// TwinCAT 3 PLC project MainPLCProject
// ProgramVersion: 3.1.4024.0
// libraries:
//   Tc2_Standard, * (Beckhoff Automation GmbH)
//   Tc2_System, * (Beckhoff Automation GmbH)
//   Tc2_TcpIp, * (Beckhoff Automation GmbH)
//   Tc2_Utilities, * (Beckhoff Automation GmbH)
//   Tc3_Module, * (Beckhoff Automation GmbH)
//   VisuDialogs, * (System)
//   VisuSymbols,3.5.10.0,System
// project tree:
//   DUTs/ ClientState.TcDUT, COM_MODE.TcDUT, DataExchangeState.TcDUT, Command.TcDUT, Message.TcDUT, MessageLogData.TcDUT, ReceiveStatus.TcDUT, SendStatus.TcDUT
//   / GlobalTextList.TcGTLO, PlcTask.TcTTO, Visualization Manager.TcVMO (not stored)
//   GVLs/ GVL.TcGVL, GVL_Constants.TcGVL
//   POUs/Classes/ ClientDataExchanger.TcPOU, COMMUNICATION.TcPOU, MESSAGE_CREATOR.TcPOU, MESSAGE_HANDLER.TcPOU, TCPClient.TcPOU
//   POUs/Helpers/ AddCounterToMessage.TcPOU, LogToWarning.TcPOU, ShiftHistoryLeft.TcPOU
//   POUs/ MAIN.TcPOU
//   VISUs/ VisualizationControlPanel.TcVIS
// real-time tasks:
//   TASK PlcTask: cycle T#10ms, priority 20, ADS port 350
//   TASK HeartbeatTask: cycle T#50000us, priority 1, ADS port 351

CONFIGURATION MainPLCProject
    RESOURCE PLC ON TwinCAT3
        TASK PlcTask(INTERVAL := T#10ms, PRIORITY := 20);
        PROGRAM MAIN WITH PlcTask : MAIN;
    END_RESOURCE
END_CONFIGURATION

// ---- DUTs/ClientState.TcDUT
{attribute 'qualified_only'}
{attribute 'strict'}
TYPE ClientState :
(
	IDLE,
	SENDING,
	RECEIVING
) := IDLE;
END_TYPE

// ---- DUTs/COM_MODE.TcDUT
{attribute 'qualified_only'}
{attribute 'strict'}
TYPE COM_MODE :
(
	Robot,
	Monarco
);
END_TYPE

// ---- DUTs/DataExchangeState.TcDUT
{attribute 'qualified_only'}
{attribute 'strict'}
TYPE DataExchangeState :
(
	IDLE,
	START,
	WORKING,
	ERROR
) := START;
END_TYPE

// ---- DUTs/Command.TcDUT
TYPE Command :
STRUCT CONSTANT
	Start : STRING(9) := 'CRISTART';
	End : STRING(7) := 'CRIEND';
	MovementVar : STRING(4) := 'VAR';
	Heartbeat : STRING(9) := 'ALIVEJOG';
	
END_STRUCT
END_TYPE

// ---- DUTs/Message.TcDUT
// Pre-made robot messages
TYPE Message :
STRUCT CONSTANT
	Connect : STRING(30) := 'CMD Connect';
	AliveDemo : STRING(63) := 'ALIVEJOG 40.0 50.0 40.0 30.0 30.0 0.0 0.0 0.0 0.0';	//Do not use, only for testing!
	EnableMessage : STRING(80) := 'CMD Enable';
END_STRUCT
END_TYPE

// ---- DUTs/MessageLogData.TcDUT
TYPE MessageLogData :
STRUCT
	systemTimeString : T_MaxString := '';
	message : STRING(GVL_Constants.MAX_RECEIVE_MESSAGE_LENGTH) := '';
END_STRUCT
END_TYPE

// ---- DUTs/ReceiveStatus.TcDUT
{attribute 'qualified_only'}
{attribute 'strict'}
TYPE ReceiveStatus :
(
	WAITING,
	RECEIVING,
	DONE,
	FAIL,
	TIMEOUT
) := RECEIVING;
END_TYPE

// ---- DUTs/SendStatus.TcDUT
{attribute 'qualified_only'}
{attribute 'strict'}
TYPE SendStatus :
(
	SENDING,
	FAIL,
	SUCCESS
) := SENDING;
END_TYPE

// ---- GVLs/GVL.TcGVL
{attribute 'qualified_only'}
VAR_GLOBAL
	// COMMUNICATION variables
	ReceivedStringArray : ARRAY[0..200] OF STRING;
	ReceivedStringWordCounter : INT := 0;

	ReceivedCMD : STRING := '';
	VarValue : STRING := '';
	VarType : STRING := '';
	VarName : STRING := '';
	//
END_VAR

// ---- GVLs/GVL_Constants.TcGVL
{attribute 'qualified_only'}
VAR_GLOBAL CONSTANT
	MAX_RECEIVE_MESSAGE_LENGTH : UDINT := 1024;
	MAX_HISTORY_SIZE : BYTE := 10;
END_VAR

// ---- POUs/MAIN.TcPOU
PROGRAM MAIN
VAR CONSTANT
	LOCAL_IP : T_IPv4Addr := '127.0.0.1';
	LOCAL_PORT : UDINT := 8080;

	REMOTE_IP : T_IPv4Addr := '192.168.3.1';
	REMOTE_PORT : UDINT := 8080;
	
	ROBOT_IP : T_IPv4Addr := '192.168.3.11';
	ROBOT_PORT : UDINT := 3920;
	
	command : Command := ();
	message : Message := ();
	//endHistoryIndex : BYTE := 9;

END_VAR
VAR
	buttonConnectPressed : BOOL;
	buttonDisconnectPressed : BOOL;	
	buttonSendPressed : BOOL;
	buttonConnectToRobotPressed : BOOL;
	buttonDebugSendPressed : BOOL;
	buttonEnableMotorsPressed : BOOL;
	
	connectTrigger : R_TRIG;
	disconnectTrigger : R_TRIG;
	sendTrigger : R_TRIG;
	connectToRobotTrigger : R_TRIG;
	debugSendTrigger : R_TRIG;
	enableMotorsTrigger : R_TRIG;
	
	client : TCPClient(LOCAL_IP, LOCAL_PORT, isEnabled := FALSE);
	LocalSystemTime : FB_LocalSystemTime;
	
	// COMMUNICATION message handling
	MessageBase : COMMUNICATION(CommunicationMODE := COM_MODE.Monarco);
	messageHandler : MESSAGE_HANDLER();
	MessageERROR : int := 0;
	//
	
	connectionMessage : STRING(20) := 'Disconnected';
	isHeartbeatEnabled : BOOL := FALSE;
	
	closeAllConnections : FB_SocketCloseALL();
	closeAll : BOOL := TRUE;	//Close all on initial startup
	
	//messageToServer : T_MaxString := 'CRISTART 1 CMD Connect CRIEND';
	messageToServer : T_MaxString := 'Hello world 2.0 CRIEND';
	debugMessageToServer : T_MaxString := 'VAR Joint 0.0 0.0 0.0 0.0 0.0 0.0 0.0 0.0 0.0';
	messageFromServer : STRING(GVL_Constants.MAX_RECEIVE_MESSAGE_LENGTH) := '';
	//finalSendMsg : STRING(100);
	
	heartbeatTimer : TON;
	heartbeatInterval : TIME := T#1S;
	
	sendCounter : INT := 1;
	finalAliveMessage : STRING(100) := '';
	totalMessagesFromServerCount : UDINT := 0;
	
	//TODO: Extract into fb? Separate task?
	currentTime : TIMESTRUCT;
	messageHistoryArray : ARRAY [0.. GVL_Constants.MAX_HISTORY_SIZE - 1] OF MessageLogData;
	currentHistoryIndex : BYTE := 0;
	currentMessageLogData : MessageLogData;
	
	//Testing
	
	executed : BOOL := FALSE;
	test : UDINT;
	test2 : UDINT;
	test3 : UDINT;

END_VAR

//On PLC reset/program download, close all connections
IF (closeAll) THEN	
	closeAll := FALSE;
	closeAllConnections(sSrvNetId := '', bExecute := TRUE, tTimeout := T#10S);
ELSE
	closeAllConnections(bExecute := FALSE);
END_IF

IF (closeAllConnections.bBusy) THEN
	RETURN;	//Do not continue the program until all connections are closed
END_IF

// === ===

// === UI Handling ===
LocalSystemTime(bEnable := TRUE, tTimeout := T#1S, systemTime => currentTime);

connectTrigger(CLK := buttonConnectPressed);
disconnectTrigger(CLK := buttonDisconnectPressed);
sendTrigger(CLK := buttonSendPressed);
connectToRobotTrigger(CLK := buttonConnectToRobotPressed);
debugSendTrigger(CLK := buttonDebugSendPressed);
enableMotorsTrigger(CLK := buttonEnableMotorsPressed);

IF (client.IsConnected) THEN
	connectionMessage := 'Connected';
ELSE
	connectionMessage := 'Disconnected';
END_IF

IF (connectTrigger.Q) THEN
	CASE MessageBase.COMMUNICATION_MODE OF
	// check for communication mode and set IP for this mode.
		COM_MODE.Robot:
			client.RemoteServerAddress := LOCAL_IP;
			client.RemoteServerPort := LOCAL_PORT;
		
		COM_MODE.Monarco:
			client.RemoteServerAddress := ROBOT_IP;
			client.RemoteServerPort := ROBOT_PORT;
	END_CASE
	client.BindReceiveMessage(variableToBind := messageFromServer);
	client.Enable();
END_IF

IF (disconnectTrigger.Q) THEN
	client.Disable();
END_IF

// === Message Sending ===
CASE MessageBase.COMMUNICATION_MODE OF
	COM_MODE.Robot:
// ROBOT COM
		IF (sendTrigger.Q) THEN  // debug: send move command to robot.
			client.Send(messageToSend := MessageBase.CREATE(COMMAND := 'VAR', COMMAND_DETAILS := 'Joint 0.0 0.0 0.0 0.0 0.0 0.0 0.0 0.0 0.0', ERROR => MessageERROR));
		END_IF

		IF (debugSendTrigger.Q) THEN // debug: not in use jet.
			client.Send(messageToSend := MessageBase.CREATE(COMMAND := '', COMMAND_DETAILS := '', ERROR => MessageERROR));
		END_IF

		IF (connectToRobotTrigger.Q) THEN
			client.Send(messageToSend := MessageBase.CREATE(COMMAND := 'CMD', COMMAND_DETAILS := 'Connect', ERROR => MessageERROR));
			isHeartbeatEnabled := TRUE;
		END_IF

		IF (enableMotorsTrigger.Q) THEN
			client.Send(messageToSend := MessageBase.CREATE(COMMAND := 'CMD', COMMAND_DETAILS := 'Enable', ERROR => MessageERROR));
		END_IF
//		
	COM_MODE.Monarco:
// MONARCO COM
		IF (sendTrigger.Q) THEN 
			client.Send(messageToSend := MessageBase.CREATE(COMMAND := 'CMD', COMMAND_DETAILS := 'LED_ON', ERROR => MessageERROR));
		END_IF

		IF (debugSendTrigger.Q) THEN
			client.Send(messageToSend := MessageBase.CREATE(COMMAND := 'CMD', COMMAND_DETAILS := 'LED_OFF', ERROR => MessageERROR));
		END_IF
//
END_CASE

// === Message Receiving ===
IF (client.NewMessageAvailable(clearFlag := TRUE)) THEN
	//Update history
	IF (currentHistoryIndex >= GVL_Constants.MAX_HISTORY_SIZE) THEN
		//Ran out of history space, discard youngest member
		currentHistoryIndex := GVL_Constants.MAX_HISTORY_SIZE;
		ShiftHistoryLeft(arr := messageHistoryArray);
	ELSE
		//Can still append
		currentHistoryIndex := currentHistoryIndex + 1;
	END_IF
	
	//Handle message
	MessageBase.HANDLE(messageFromServer);
	
	//Add new entry
	currentMessageLogData.message := messageFromServer;	
	currentMessageLogData.systemTimeString := SYSTEMTIME_TO_STRING(in := currentTime);
	messageHistoryArray[currentHistoryIndex - 1] := currentMessageLogData;
END_IF
// === ===

// === Heartbeat ===
heartbeatTimer(IN := isHeartbeatEnabled, PT := heartbeatInterval);

IF (heartbeatTimer.Q AND client.IsClientEnabled) THEN
	heartbeatTimer(IN := FALSE);
	client.Send(messageToSend := MessageBase.CREATE('ALIVEJOG', '40.0 50.0 40.0 30.0 30.0 0.0 0.0 0.0 0.0', ERROR => MessageERROR));
END_IF
// === ===

client(totalMessagesReceived => totalMessagesFromServerCount);

END_PROGRAM

// ---- POUs/Classes/TCPClient.TcPOU
FUNCTION_BLOCK TCPClient
VAR CONSTANT
	CLIENT_RECONNECT_TIME : TIME := T#31S;
	MAX_MESSAGE_LENGTH : INT := 255;
	MAX_RECEIVE_MESSAGE_LENGTH : UDINT := GVL_Constants.MAX_RECEIVE_MESSAGE_LENGTH;
END_VAR
VAR_OUTPUT
	totalMessagesReceived : UDINT := 0;
END_VAR
VAR
	m_isClientEnabled : BOOL := TRUE;	
	m_serverNetID : STRING(80) := '';
	
	ClientServerConnection : FB_ClientServerConnection;
	SocketSend : FB_SocketSend;
	SocketReceive : FB_SocketReceive;
	m_clientDataExchanger : ClientDataExchanger;	//Note implemented yet: leave for later, use as
	m_socketHandle : T_HSOCKET;
	
	
	m_remoteServerAddress : T_IPv4Addr;	
	m_remoteServerPort : UDINT := 0;
	
	//Note: make it an input and send only when the class is called?
	m_messageToSend : T_MaxString := 'Hello world!';
	//m_messageReceived : T_MaxString;	// The latest message received from the server //TODO: REMOVE, Depricated
	m_messageReceivedRef : REFERENCE TO STRING(MAX_RECEIVE_MESSAGE_LENGTH);
	
	m_isConnected : BOOL := FALSE;
	m_isBusy : BOOL;
	m_errorOccured : BOOL;
	m_lastErrorId : UDINT;
	
	
	m_currentSocketState : Tc2_TcpIp.E_SocketConnectionState;
	m_currentState : ClientState := ClientState.RECEIVING;	

	m_sendDataExchangeState : DataExchangeState := DataExchangeState.START;	
	m_sendRequested: BOOL;
	m_sendStatus : SendStatus;
	m_sendErrorId : UDINT;
	m_sendTimeout : TIME := T#15S;	//Note: Lower?
	
	//Receiving
	m_receiveDataExchangeState : DataExchangeState := DataExchangeState.IDLE;	
	m_isReceiveTimerEnabled : BOOL := TRUE;
	m_receiveTimer : TON();
	m_isReceiveTimeoutEnabled : BOOL := FALSE;	
	m_receiveTimeoutTimer : TON();
	m_receiveBuffer : STRING(MAX_RECEIVE_MESSAGE_LENGTH) := '';
	m_totalBytesReceived : UDINT := 0;
	m_receiveTimeout : TIME := T#1M;
	m_readInterval : TIME := T#10MS;
//	m_receiveMessageDelimiter : BYTE := F_ToASC(';');	//Note: Use plain 0 (without F_ToASC()) for \0
	m_receiveMessageDelimiter : BYTE := 0;	//'\0'	//Not used currently
	m_delimiterString : STRING(80) := 'CRIEND';	//TODO: Make settable via property
	m_receivedMessage : T_MaxString := '';
	m_receiveStatus : ReceiveStatus;
	m_newDataAvailable : BOOL := FALSE;	//Reset to false when it is read
	m_receiveErrorId : UDINT := 0;
	m_totalMessagesReceived : UDINT := 0;
END_VAR

//Handler code
//Does that need to be executed every cycle or can I put it in eSOCKET_DISCONNECTED state?
ClientServerConnection(sSrvNetID := m_serverNetID,
						 nMode := 0,
						 sRemoteHost := RemoteServerAddress,
						 nRemotePort := m_remoteServerPort,
						 tReconnect := CLIENT_RECONNECT_TIME,
						 bEnable := IsClientEnabled,
						 bBusy => m_isBusy,
						 bError => m_errorOccured,
						 nErrId => m_lastErrorId,
						 hSocket => m_socketHandle,
						 eState => m_currentSocketState);

CASE m_currentSocketState OF
	E_SocketConnectionState.eSOCKET_DISCONNECTED:
		m_isConnected := FALSE;
	//
	E_SocketConnectionState.eSOCKET_SUSPENDED:
	//Change from disconnected to connected or vise versa
		m_isConnected := FALSE;
	//
	E_SocketConnectionState.eSOCKET_CONNECTED:
		m_isConnected := TRUE;
END_CASE

IF (NOT m_isConnected) THEN
	RETURN;
END_IF

// Executed only if a connection is established

CASE m_currentState OF
	//
	ClientState.SENDING:
		m_sendStatus := SendMessage(messageToSend := m_messageToSend, timeout := m_sendTimeout, errorId => m_sendErrorId);
		IF (m_sendStatus = SendStatus.SUCCESS) THEN
			m_currentState := ClientState.RECEIVING;
		ELSIF (m_sendStatus = SendStatus.FAIL) THEN
			//Sending failed
			ADSLOGDINT(msgCtrlMask := ADSLOG_MSGTYPE_WARN, msgFmtStr := 'Send fail error: %d', dintArg := UDINT_TO_DINT(m_sendErrorId));
			m_currentState := ClientState.RECEIVING;
		END_IF
		
	//
	ClientState.RECEIVING:
		m_receiveStatus := Receive(timeout := m_receiveTimeout, 
									readInterval := m_readInterval, 
									messageDelimiter := m_receiveMessageDelimiter,	//Currently not used
									errorId => m_receiveErrorId);
		
		IF (m_receiveStatus <> ReceiveStatus.RECEIVING) THEN
			IF (m_receiveStatus = ReceiveStatus.DONE) THEN
				//
				totalMessagesReceived := totalMessagesReceived + 1;
				m_newDataAvailable := TRUE;
			END_IF
			
			IF (m_receiveStatus = ReceiveStatus.FAIL) THEN
				//Fail Handling
				LogToWarning(msgFmtStr := 'Receive fail error: %s', messageArg := UDINT_TO_STRING(m_receiveErrorId));
			END_IF
			
			IF (m_receiveStatus = ReceiveStatus.TIMEOUT) THEN
				//Timeout handling
				LogToWarning(msgFmtStr := 'Receive timed out', messageArg := '');
				//Disable();	//Disable on timeout
			END_IF
	
			IF (m_sendRequested) THEN
				m_sendRequested := FALSE;
				m_sendErrorId := 0;
				m_currentState := ClientState.SENDING;
			END_IF
		END_IF						
	
	// After done receiving, go to idle?
	//
END_CASE

METHOD PUBLIC BindReceiveMessage : BOOL
VAR_INPUT
	variableToBind : REFERENCE TO STRING(MAX_RECEIVE_MESSAGE_LENGTH);
END_VAR
m_messageReceivedRef REF= variableToBind;
END_METHOD

METHOD PUBLIC Disable : BOOL
m_isClientEnabled := False;
END_METHOD

METHOD PUBLIC Enable : BOOL
VAR_INPUT
END_VAR
m_isClientEnabled := TRUE;
END_METHOD

METHOD FB_init : BOOL
VAR_INPUT
	bInitRetains : BOOL; // if TRUE, the retain variables are initialized (warm start / cold start)
	bInCopyCode : BOOL;  // if TRUE, the instance afterwards gets moved into the copy code (online change)
	
	remoteServerAddress : T_IPv4Addr := '127.0.0.1';
	remoteServerPort : UDINT := 8080;
	isEnabled : BOOL := FALSE;
END_VAR
m_remoteServerAddress := remoteServerAddress;
m_remoteServerPort := remoteServerPort;
m_isClientEnabled := isEnabled;
END_METHOD

PROPERTY IsClientEnabled : BOOL
GET
IsClientEnabled := m_isClientEnabled;
END_GET
END_PROPERTY

PROPERTY IsConnected : BOOL
GET
IsConnected := m_isConnected;
END_GET
END_PROPERTY

PROPERTY LastSendStatus : SendStatus
GET
LastSendStatus := m_sendStatus;
END_GET
END_PROPERTY

METHOD PUBLIC NewMessageAvailable : BOOL
VAR_INPUT
	clearFlag : BOOL := FALSE;	//Clears the new message flag if set to true, does not otherwise
END_VAR
NewMessageAvailable := m_newDataAvailable;

IF (clearFLag) THEN
	m_newDataAvailable := FALSE;
END_IF
END_METHOD

METHOD PRIVATE Receive : ReceiveStatus
VAR_INPUT
	timeout : TIME := T#10S;
	readInterval : TIME := T#10MS;
	messageDelimiter : BYTE := 0;
END_VAR

VAR_OUTPUT
	errorId : UDINT;
END_VAR

VAR
	errorOccurred : BOOL;	//can sty
	isBusy : BOOL;	//can stay																
	
	timedout : BOOL := FALSE;	//Output of TON
	receivedBytes : UDINT := 0;	//Output, should be fine to be here
	
	startPosition : UDINT := 0;	//Can stay, assigned before used
	endPosition : UDINT := 0;	//Can stay, assigned before used
	currentFrameLength : UDINT := 0; // Length of string received this cycle	//Should be fine
	posOfDelimiter : UDINT := 0;
	
	
	index : UDINT := 0;	//For-loop index
	
END_VAR
m_receiveTimer(IN := m_isReceiveTimerEnabled);
m_receiveTimeoutTimer(IN := m_isReceiveTimeoutEnabled, PT := timeout, Q => timedout);

CASE m_receiveDataExchangeState OF
	DataExchangeState.IDLE:
		//Reset variables
		m_isReceiveTimerEnabled := FALSE;
		m_receiveTimer(IN := m_isReceiveTimerEnabled, PT := T#0MS); 	//Do not wait for the first read
		m_isReceiveTimeoutEnabled := FALSE;
		Receive := ReceiveStatus.WAITING;
		m_receiveDataExchangeState := DataExchangeState.START;
	//
	DataExchangeState.START:
		Receive := ReceiveStatus.WAITING;
		m_isReceiveTimerEnabled := TRUE;
		IF (m_receiveTimer.Q) THEN
			SocketReceive(bExecute := FALSE);
			SocketReceive(sSrvNetId := m_serverNetID,
						  hSocket := m_socketHandle,
						  pDest := ADR(m_receiveBuffer) + m_totalBytesReceived,
						  cbLen := SIZEOF(m_receiveBuffer) - m_totalBytesReceived,
						  tTimeout := timeout,
						  bExecute := TRUE);	
			
			m_receiveDataExchangeState := DataExchangeState.WORKING;
		END_IF
	//
	DataExchangeState.WORKING:
		Receive := ReceiveStatus.RECEIVING;
		SocketReceive(bExecute := FALSE,
				tTimeout := timeout,
				bBusy => isBusy,
				bError => errorOccurred,
				nErrId => errorId,
				nRecBytes => receivedBytes);
		//Enable timeout
		IF (NOT isBusy AND NOT errorOccurred) THEN
			IF (receivedBytes > 0) THEN
				startPosition := m_totalBytesReceived;
				//Calculate new total
				m_totalBytesReceived := m_totalBytesReceived + receivedBytes;
				endPosition := m_totalBytesReceived - 1;
				currentFrameLength := 0;
				//Only proceed if we have enough space
				IF (m_totalBytesReceived < SIZEOF(m_messageReceivedRef)) THEN
					m_receiveTimer (PT := T#0MS); //Read asap
					//Bytes received, disable timeout check
					m_isReceiveTimeoutEnabled := FALSE;
					//Search for end of message delimiter
					posOfDelimiter := INT_TO_UDINT(FIND(STR1 := m_receiveBuffer, STR2 := m_delimiterString));
					
					IF (posOfDelimiter = 0) THEN
						//Delimiter not found
						LogToWarning('Delim not found', '');
						RETURN;
					END_IF
					
					currentFrameLength := posOfDelimiter + 6{delimiter size} - 1;
					MEMCPY(destAddr := ADR(m_messageReceivedRef), srcAddr := ADR(m_receiveBuffer), n := currentFrameLength);
					MEMSET(destAddr := ADR(m_receiveBuffer), fillByte := 0, n := SIZEOF(m_receiveBuffer));	//Clear buffer
					m_totalBytesReceived := 0;
					
					//All received
					Receive := ReceiveStatus.DONE;
					m_receiveDataExchangeState := DataExchangeState.IDLE;
					//OLD Find TODO: Find a way to implement via a function? So that you can use both
//					FOR index := startPosition TO endPosition BY 1 DO
//						IF (m_receiveBuffer[index] = messageDelimiter) THEN	//End of message check
//							//End of message received
//							currentFrameLength := index + 1;
							
//							MEMCPY(destAddr := ADR(m_messageReceivedRef), srcAddr := ADR(m_receiveBuffer), n := currentFrameLength);
//							//Move the remaining data bytes to the begining
//							MEMMOVE(ADR(m_receiveBuffer), ADR(m_receiveBuffer[currentFrameLength]), m_totalBytesReceived - currentFrameLength); 
//							//Recalculate remaining data byte length
//							m_totalBytesReceived := m_totalBytesReceived - currentFrameLength;
//							//All received
//							Receive := ReceiveStatus.DONE;
//							m_receiveDataExchangeState := DataExchangeState.IDLE;
//							EXIT;
//						END_IF
//					END_FOR

				ELSE	
					//No more space in the receive object
					Receive := ReceiveStatus.FAIL;
					m_receiveDataExchangeState := DataExchangeState.ERROR;
				END_IF //IF (totalBytesReceived < SIZEOF(receivedMessage))
			ELSE
				//No bytes received
				m_receiveTimer (PT := readInterval);
				m_isReceiveTimeoutEnabled := TRUE;
				
				//IF (timedout) THEN
				IF (m_receiveTimeoutTimer.Q) THEN
					Receive := ReceiveStatus.TIMEOUT;
					m_receiveDataExchangeState := DataExchangeState.ERROR;
				ELSE
					//Read again
					m_receiveDataExchangeState := DataExchangeState.START;
				END_IF
			END_IF //IF (receivedBytes > 0)
		
		ELSIF (errorOccurred) THEN
			Receive := ReceiveStatus.FAIL;
			m_receiveDataExchangeState := DataExchangeState.ERROR;
		END_IF	//IF (NOT isBusy AND NOT errorOccurred)
		
	//
	DataExchangeState.ERROR:
		//Variable resets in case of an error
		m_totalBytesReceived := 0;	//Reset counter
		m_receiveBuffer := DELETE(STR := m_receiveBuffer, POS := 1, LEN := 255);	//Reset receive buffer
		m_receiveDataExchangeState := DataExchangeState.IDLE;
	//
END_CASE
END_METHOD

//Note: After reading, NewDataAvailable returns false until new data arrives
PROPERTY ReceivedData : T_MaxString
GET
ReceivedData := m_receivedMessage;
m_newDataAvailable := FALSE;
END_GET
END_PROPERTY

PROPERTY RemoteServerAddress : T_IPv4Addr
GET
RemoteServerAddress := m_remoteServerAddress;
END_GET
SET
m_remoteServerAddress := RemoteServerAddress;
END_SET
END_PROPERTY

PROPERTY RemoteServerPort : UDINT
GET
RemoteServerPort := m_remoteServerPort;
END_GET
SET
m_remoteServerPort := RemoteServerPort;
END_SET
END_PROPERTY

METHOD Send : BOOL
VAR_INPUT
	messageToSend : T_MaxString;
END_VAR
m_sendRequested := TRUE;
m_messageToSend := messageToSend;
END_METHOD

//Wrapper for SocketSend. On error, check the errorId variable
METHOD PRIVATE SendMessage : SendStatus
VAR_INPUT
	messageToSend : T_MaxString;
	timeout : TIME;
END_VAR

VAR_OUTPUT
	errorId : UDINT := 0;
END_VAR

VAR
	errorOccurred : BOOL;	
	isBusy : BOOL;	
END_VAR
CASE m_sendDataExchangeState OF
	DataExchangeState.START:
		errorId := 0;
		
		SocketSend(sSrvNetId := m_serverNetID,
				   hSocket := m_socketHandle,
				   cbLen := INT_TO_UDINT(LEN(messageToSend) + 1),
		   		   pSrc := ADR(messageToSend),
				   tTimeout := timeout,
				   bExecute := FALSE
				   );

		m_sendDataExchangeState := DataExchangeState.WORKING;
	//
	DataExchangeState.WORKING:
		
		SocketSend(bExecute := TRUE,
				   bError => errorOccurred,
		   		   nErrId => errorId,
		   		   bBusy => isBusy);
		
		IF (NOT isBusy AND NOT errorOccurred) THEN
			SendMessage := SendStatus.SUCCESS;
			m_sendDataExchangeState := DataExchangeState.START;
		ELSIF (errorOccurred) THEN
			SendMessage := SendStatus.FAIL;
			m_sendDataExchangeState := DataExchangeState.START;
		ELSIF (isBusy) THEN
			SendMessage := SendStatus.SENDING;
		END_IF 
	//
END_CASE
END_METHOD

END_FUNCTION_BLOCK

// ---- POUs/Classes/ClientDataExchanger.TcPOU
FUNCTION_BLOCK ClientDataExchanger
VAR_INPUT
END_VAR
VAR_OUTPUT
END_VAR
VAR
	//TODO: Finish https://infosys.beckhoff.com/english.php?content=../content/1033/tf6310_tc3_tcpip/84203915.html&id=
	//Note: Needed? Wouldn't it be better to just have a .Send and .Receive methods?
	m_socketHandle : T_HSOCKET;
	m_messageToServer : T_MaxString;	

END_VAR

END_FUNCTION_BLOCK

// ---- POUs/Helpers/LogToWarning.TcPOU
FUNCTION LogToWarning : BOOL
VAR_INPUT
	msgFmtStr : T_MaxString;
	messageArg : T_MaxString;
END_VAR
VAR
END_VAR

ADSLOGSTR(msgCtrlMask := ADSLOG_MSGTYPE_WARN, msgFmtStr := msgFmtStr, strArg := messageArg);

END_FUNCTION

// ---- POUs/Classes/COMMUNICATION.TcPOU
FUNCTION_BLOCK COMMUNICATION
VAR_INPUT
	
END_VAR
VAR_OUTPUT
END_VAR
VAR
	m_COMMUNICATION_MODE : COM_MODE;
	messageCreator : MESSAGE_CREATOR('CRISTART', 'CRIEND', 1);
	messageHandler : MESSAGE_HANDLER();
END_VAR

PROPERTY PUBLIC COMMUNICATION_MODE : COM_MODE
GET
COMMUNICATION_MODE := m_COMMUNICATION_MODE;
END_GET
SET
m_COMMUNICATION_MODE := COMMUNICATION_MODE;
END_SET
END_PROPERTY

METHOD PUBLIC CREATE : STRING
VAR_INPUT
	COMMAND : STRING;
	COMMAND_DETAILS : STRING;
END_VAR
VAR_OUTPUT
	ERROR : INT := 0;
END_VAR
IF (COMMUNICATION_MODE = COM_MODE.Robot) THEN 
	// creates string for robot when in Robot mode
	CREATE := MessageCreator.ROBOT_MESSAGE(COMMAND, COMMAND_DETAILS, ERROR => ERROR);
ELSIF (COMMUNICATION_MODE = COM_MODE.Monarco) THEN 
	// creates string for monarco when in Monarco mode
	CREATE := MessageCreator.MONARCO_MESSAGE_CMD(COMMAND_DETAILS, ERROR => ERROR);
			// JUST THE CMD MONARCO MESSAGE FOR NOW!!
END_IF
END_METHOD

METHOD FB_init : BOOL
VAR_INPUT
	bInitRetains : BOOL; // if TRUE, the retain variables are initialized (warm start / cold start)
	bInCopyCode : BOOL;  // if TRUE, the instance afterwards gets moved into the copy code (online change)
	
	communicationMODE : COM_MODE;
END_VAR
COMMUNICATION_MODE := communicationMode;
END_METHOD

METHOD PUBLIC HANDLE : INT
VAR_INPUT
	FULL_STRING : STRING;
END_VAR
IF (COMMUNICATION_MODE = COM_MODE.Robot) THEN 
	// handles string from robot when in Robot mode (RECEIVE_ROBOT())
	MessageHandler.RECEIVE_ROBOT(FULL_STRING, ERROR => HANDLE);
ELSIF (COMMUNICATION_MODE = COM_MODE.Monarco) THEN 
	// handles string from monarco when in Monarco mode (RECEIVE_MONARCO())
	MessageHandler.RECEIVE_MONARCO(FULL_STRING, ERROR => HANDLE);
END_IF
END_METHOD

END_FUNCTION_BLOCK

// ---- POUs/Classes/MESSAGE_CREATOR.TcPOU
FUNCTION_BLOCK PUBLIC MESSAGE_CREATOR
VAR_INPUT
END_VAR
VAR_OUTPUT
END_VAR
VAR
	m_START_COMMAND : STRING;
	m_END_COMMAND : STRING;
	m_MESSAGE_COUNT : INT;
END_VAR

PROPERTY PUBLIC END_COMMAND : STRING
GET
END_COMMAND := m_END_COMMAND;
END_GET
SET
m_END_COMMAND := END_COMMAND;
END_SET
END_PROPERTY

METHOD FB_init : BOOL
VAR_INPUT
	bInitRetains : BOOL; // if TRUE, the retain variables are initialized (warm start / cold start)
	bInCopyCode : BOOL;  // if TRUE, the instance afterwards gets moved into the copy code (online change)
	
	STARTcommand : STRING;
	ENDcommand : STRING;
	MESSAGEcount : INT;
END_VAR
START_COMMAND := STARTcommand;
END_COMMAND := ENDcommand;
MESSAGE_COUNT := MESSAGEcount;
END_METHOD

PROPERTY PUBLIC MESSAGE_COUNT : INT
GET
MESSAGE_COUNT := m_MESSAGE_COUNT;
END_GET
SET
m_MESSAGE_COUNT := MESSAGE_COUNT;
END_SET
END_PROPERTY

METHOD PUBLIC MONARCO_MESSAGE_CMD : STRING
VAR_INPUT
	COMMAND_DETAILS : STRING;
END_VAR
VAR CONSTANT
	COMMAND : STRING := 'CMD';
	SEPARATOR : STRING := ' ';
END_VAR
VAR_OUTPUT
	ERROR : INT := 0;
END_VAR
IF (COMMAND_DETAILS <> '') THEN // if command_details is not empty, create command string.
	MONARCO_MESSAGE_CMD := 
		CONCAT(COMMAND, 
		CONCAT(SEPARATOR, 
			COMMAND_DETAILS));
			
ELSE // else return error string and error code 1.
	MONARCO_MESSAGE_CMD := 'ERROR_NoCommandDetailsGiven';
	ERROR := 1;
END_IF

//FULL_MONARCO_CMD_MESSAGE := 'CMD TURN_LED_ON';
END_METHOD

METHOD PUBLIC MONARCO_MESSAGE_VAR : STRING
VAR_INPUT
	VARIABLE_NAME : STRING;
	VARIABLE_TYPE : STRING;
	VARIABLE_VALUE : STRING;
END_VAR
VAR CONSTANT
	COMMAND : STRING := 'VAR';
	SEPARATOR : STRING := ' ';
END_VAR
VAR_OUTPUT
	ERROR : INT := 0;
END_VAR
IF (VARIABLE_NAME <> '' AND VARIABLE_TYPE <> '' AND VARIABLE_VALUE <> '') THEN 
	// if all values given, create var string.
	MONARCO_MESSAGE_VAR := 
			CONCAT(COMMAND, 
			CONCAT(SEPARATOR, 
			CONCAT(VARIABLE_NAME,
			CONCAT(SEPARATOR, 
			CONCAT(VARIABLE_TYPE,
			CONCAT(SEPARATOR, 
				VARIABLE_VALUE))))));
				
ELSE // else return error string, and error code 1.
	MONARCO_MESSAGE_VAR := 'ERROR_SomeValuesMissing';
	ERROR := 1;
END_IF

//FULL_MONARCO_VAR_MESSAGE := 'CMD varName1 INT 9';
END_METHOD

METHOD PUBLIC ROBOT_MESSAGE : T_MaxString
VAR_INPUT
	COMMAND : STRING;
	COMMAND_DETAILS : STRING;
END_VAR
VAR_OUTPUT
	ERROR : INT := 0;
END_VAR
 // CREATES A STRING THAT THE IGUS ROBOT CAN READ AND UNDERSTAND VIA ETHERNET.
ROBOT_MESSAGE := 
CONCAT(START_COMMAND, 
CONCAT(' ', 
CONCAT(INT_TO_STRING(MESSAGE_COUNT), 
CONCAT(' ', 
CONCAT(COMMAND, 
CONCAT(' ', 
CONCAT(COMMAND_DETAILS, 
CONCAT(' ', END_COMMAND))))))));

MESSAGE_COUNT := (MESSAGE_COUNT MOD 9999)+ 1;

//FULL_ROBOT_MESSAGE := 'CRISTART 1 CMD Connect CRIEND';
END_METHOD

PROPERTY PUBLIC START_COMMAND : STRING
GET
START_COMMAND := m_START_COMMAND;
END_GET
SET
m_START_COMMAND := START_COMMAND;
END_SET
END_PROPERTY

END_FUNCTION_BLOCK

// ---- POUs/Classes/MESSAGE_HANDLER.TcPOU
FUNCTION_BLOCK PUBLIC MESSAGE_HANDLER
VAR_INPUT
END_VAR
VAR_OUTPUT
END_VAR
VAR
END_VAR

METHOD FB_init : BOOL
VAR_INPUT
	bInitRetains : BOOL; // if TRUE, the retain variables are initialized (warm start / cold start)
	bInCopyCode : BOOL;  // if TRUE, the instance afterwards gets moved into the copy code (online change)

	
END_VAR
END_METHOD

METHOD PUBLIC RECEIVE_MONARCO : INT
VAR_INPUT
	FULL_STRING : STRING;
END_VAR
VAR
	FOUND_SEPARATOR : BOOL;
	COMMAND_CMD : STRING := 'CMD';
	COMMAND_VAR : STRING := 'VAR';
	count : INT := 0;
	MESSAGE_ARRAY : ARRAY[1..4] OF STRING;
	
	SeparatorChar : STRING := ' ';
	tempString : STRING := '';
	stringLeft : STRING := '';
	stringLeftSize : UDINT := 999;
	stringRight : STRING := '';
	stringRightSize : UDINT := 999;
END_VAR
VAR_OUTPUT
	ERROR : INT := 0;
END_VAR
// save received string into changeble variable.

tempString := FULL_STRING;

FOR count := 1 TO 4 BY 1 DO
	FOUND_SEPARATOR := FindAndSplitChar(
		sSeparatorChar := SeparatorChar, 	// split when this char found
		pSrcString := ADR(tempString), 		// string that will be split
		pLeftString := ADR(stringLeft), 	// first string (left) (FIRST WORD)
		nLeftSize := stringLeftSize, 		// first string size (right)
		pRightString := ADR(stringRight), 	// second string (right) (REST OF STRING)
		nRightSize := stringRightSize, 		// second string size (right)
		bSearchFromright := FALSE);			// when false start searching from the left
		
	IF FOUND_SEPARATOR THEN
		MESSAGE_ARRAY[count] := stringLeft; // saving the left string in message_array.
		tempString := stringRight; // saving the rest of the string for the next split.
	ELSE // ERROR: the separator char could not be found.
		MESSAGE_ARRAY[count] := tempString; // saving the string in case it was the last word.
		ERROR := count; 
		count := 10;
	END_IF
END_FOR

IF (ERROR = 2 OR ERROR = 4) THEN // handle message_array when CMD or VAR was the command.
	ERROR := 0;
	IF (MESSAGE_ARRAY[1] = COMMAND_CMD) THEN // when CMD was the command.
		GVL.ReceivedCMD := MESSAGE_ARRAY[2];
	ELSIF (MESSAGE_ARRAY[1] = COMMAND_VAR) THEN // when VAR was the command.
		GVL.VarName := MESSAGE_ARRAY[2];
		GVL.VarType := MESSAGE_ARRAY[3];
		GVL.VarValue := MESSAGE_ARRAY[4];
	ELSE
		ERROR := 5; // ERROR: neither CMD or VAR was red.
	END_IF
END_IF
END_METHOD

METHOD PUBLIC RECEIVE_ROBOT : INT
VAR_INPUT
	FULL_STRING : STRING;
END_VAR
VAR
	tempString : STRING;
	SeparatorChar : STRING := ' ';
	stringLeft : STRING;
	stringLeftSize : UDINT := 999;
	stringRight : STRING;
	stringRightSize : UDINT := 999;
	foundSeparator : BOOL;
	
	stepCount : INT;
END_VAR
VAR_OUTPUT
	ERROR : INT;
END_VAR
tempString := FULL_STRING;
FOR stepCount := 0 TO 200 BY 1 DO
	foundSeparator := FindAndSplitChar( // SEPERATE THE STRING, FIRST WORD -- REST OF STRING
		sSeparatorChar := SeparatorChar, 	// split when this char found
		pSrcString := ADR(tempString), 		// string that will be split
		pLeftString := ADR(stringLeft), 	// first string (left) (FIRST WORD)
		nLeftSize := stringLeftSize, 		// first string size (right)
		pRightString := ADR(stringRight), 	// second string (right) (REST OF STRING)
		nRightSize := stringRightSize, 		// second string size (right)
		bSearchFromright := FALSE);			// when false start searching from the left
	IF (stringRight = 'CRIEND') THEN // CHECK FOR ENDING
		GVL.ReceivedStringArray[stepCount] := stringLeft;
		GVL.ReceivedStringArray[stepCount + 1] := stringRight;
		GVL.ReceivedStringWordCounter := (stepCount + 1);
		stepCount := 210;
		ERROR := 0;
	ELSE // OTHERWISE SAVE SEPPERATED VAR AND CONTINUE
		IF (foundSeparator) THEN // CHECK FOR ERROR
			tempString := stringRight;
			GVL.ReceivedStringArray[stepCount] := stringLeft;
		ELSE // ERROR OCCURED, COULD NOT FIND SEPARATOR
			stepCount := 210;
			ERROR := 3;
		END_IF 
	END_IF 
END_FOR
END_METHOD

END_FUNCTION_BLOCK

// ---- POUs/Helpers/ShiftHistoryLeft.TcPOU
FUNCTION ShiftHistoryLeft : BOOL
VAR_INPUT
	//TODO: Use constant in GVL_Constants
	arr : REFERENCE TO ARRAY[0..9] OF MessageLogData;
END_VAR
VAR
	i : INT := 0;
END_VAR

FOR i:= 0 TO 9 - 1 BY 1 DO
	arr[i] := arr[i + 1];
END_FOR

END_FUNCTION

// ---- POUs/Helpers/AddCounterToMessage.TcPOU
FUNCTION AddCounterToMessage : T_MaxString
VAR_INPUT
	counter : INT;
	message : T_MaxString;
END_VAR
VAR
END_VAR

AddCounterToMessage := CONCAT('CRISTART ', 
					   CONCAT(INT_TO_STRING(counter), 
					   CONCAT(' ',
					   CONCAT(message, 
							 ' CRIEND'))));

END_FUNCTION

// ---- GlobalTextList.TcGTLO
TEXTLIST GlobalTextList
  423 = 'Connect'
  286 = 'Connect To Robot'
  403 = 'Debug Send'
  428 = 'Disconnect'
  622 = 'Enable Motors'
  229 = 'History'
  290 = 'Message'
  597 = 'Messages received: %d'
  193 = 'Receive History'
  729 = 'Send'
  222 = 'Server: %s'
  529 = 'Status: %s'
  256 = 'Time'
END_TEXTLIST

// ---- VISUs/VisualizationControlPanel.TcVIS
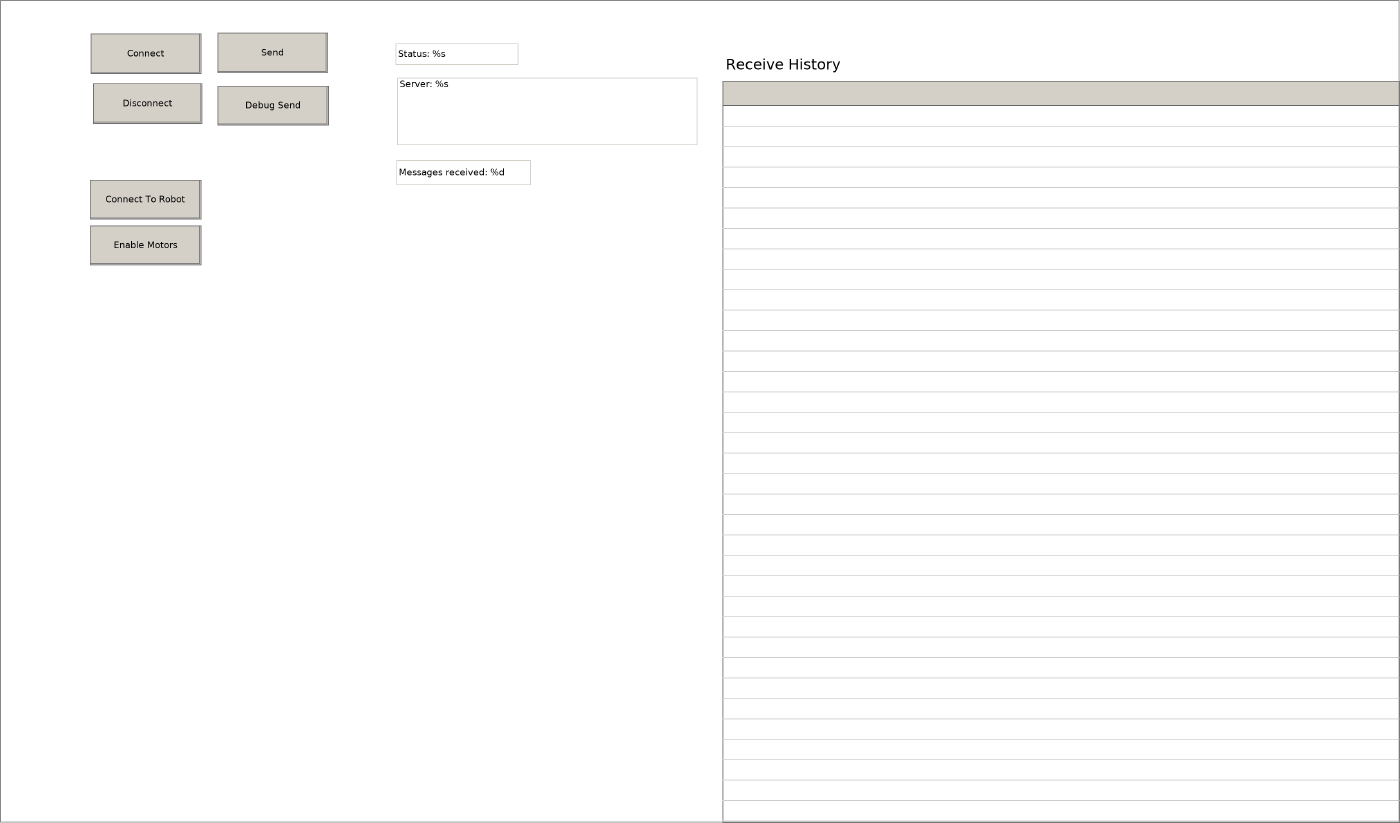
VISUALIZATION VisualizationControlPanel  // 1713x1007
    Button (114,102 133x49), "Disconnect"
        tap MAIN.buttonDisconnectPressed
    Button (266,40 135x49), "Send"
        tap MAIN.buttonSendPressed
    Button (111,41 135x49), "Connect"
        tap MAIN.buttonConnectPressed
    Textfield (486,95 367x82), "Server: %s", text variable: MAIN.messageFromServer
    Textfield (485,196 164x30), "Messages received: %d", text variable: MAIN.totalMessagesFromServerCount
    Table (884,99 829x908), data array: MAIN.messageHistoryArray
        p3854506369: MAIN.messageHistoryArray[INDEX].systemTimeString
        p1892666644: MAIN.messageHistoryArray[INDEX].message
        p511219082: Message
    Label (885,64 182x30), "Receive History"
    Button (110,220 136x48), "Connect To Robot"
        tap MAIN.buttonConnectToRobotPressed
    Button (266,105 136x48), "Debug Send"
        tap MAIN.buttonDebugSendPressed
    Button (110,276 136x48), "Enable Motors"
        tap MAIN.buttonEnableMotorsPressed
    Textfield (484,53 150x26), "Status: %s", text variable: MAIN.connectionMessage
END_VISUALIZATION
